// TwinCAT 3 PLC project PLC1
// ProgramVersion: 3.1.4026.24
// libraries:
//   AdsGamepad, * (Beckhoff Community)
//   Tc2_Standard, * (Beckhoff Automation GmbH)
//   Tc2_System, * (Beckhoff Automation GmbH)
//   Tc3_Module, * (Beckhoff Automation GmbH)
// project tree:
//   / PlcTask.TcTTO (not stored)
//   POUs/ MAIN.TcPOU
// real-time tasks:
//   TASK PlcTask: cycle T#10ms, priority 20, ADS port 351

// ---- POUs/MAIN.TcPOU
PROGRAM MAIN
VAR
	// Gamepad from the AdsGamepad library. An empty NetID means the local machine
	Gamepad			: FB_Gamepad_Controller('', 1);
	bEnableMover	: BOOL := TRUE;

	// Raw stick values. Mapping them onto axes or movers is application code
	fStickX			: LREAL;
	fStickY			: LREAL;
END_VAR

Gamepad.Cycle();

// Read the left stick. The jog helper FBs are gone from the library, so how these
// values drive an axis or a mover is up to the application. See MIGRATION.md
fStickX := Gamepad.P_Left_Joystick.fX;
fStickY := Gamepad.P_Left_Joystick.fY;

END_PROGRAM
